{attribute 'GeneratedUsingTerminal: EPP1816-0003-0016'}
{attribute addProperty BoxType "EPP1816-0003-0016"}
{attribute addProperty Id "InputAT %I*ARRAY[0..7] OF BOOL8Sync_errorAT %I*BOOL1TxPDO_ToggleAT %I*BOOL1"}
{attribute addProperty CRC "780220065"}
{attribute addProperty Size "10"}
TYPE DIG_Inputs_Channel_ACAA0425 :
STRUCT
	{attribute addProperty Name "Input"}
	Input AT %I* : ARRAY[0..7] OF BOOL;
	{attribute addProperty Name "Sync_error"}
	Sync_error AT %I* : BOOL;
	{attribute addProperty Name "TxPDO_Toggle"}
	TxPDO_Toggle AT %I* : BOOL;
END_STRUCT
END_TYPE

(* stored: Version 1.2.0.0, ProductVersion 3.1.4024.9
   DUT DIG_Inputs_Channel_ACAA0425: Id {d8ae51f7-27ca-4f8d-b222-aca0e8ded6df} *)
